FUNCTION F_Return : REAL
VAR_INPUT
    fIn : REAL;
END_VAR

F_Return := fIn;

END_FUNCTION

(* stored: Version 1.1.0.1
   POU F_Return: Id {11111111-1111-1111-1111-111111111105} *)
